TYPE ForceLimiterFsmState :
(
	FsmState_Idle := 0,
	FsmState_Rih,
	FsmState_Pooh,
	NUM_FsmStates
)BYTE;
END_TYPE

(* stored: Version 1.1.0.1, ProductVersion 3.1.4024.6
   DUT ForceLimiterFsmState: Id {d0a762da-cae6-484e-b06a-41a112a4ee36} *)
